(* PLC project Unnamed, Unknown Unnamed 1 *)
(* stored: creationDateTime 2024-10-03T07:22:18, modificationDateTime 2024-10-03T07:23:21 *)

PROGRAM program0
  VAR
    TON0 : TON;
  END_VAR

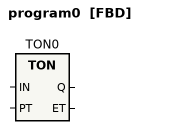
(* FBD diagram, written out as Structured Text *)
TON0();
END_PROGRAM

CONFIGURATION Config0
  RESOURCE Res0 ON PLC
    TASK task0(INTERVAL := T#20ms, PRIORITY := 0);
    PROGRAM instance0 WITH task0 : program0;
  END_RESOURCE
END_CONFIGURATION
